TYPE ST_Software_Info :
STRUCT
	sTwinCATVersion		: STRING;
	iADSPort			: UINT;
	sProjectName		: STRING;
	sAppTimeStamp		: DATE_AND_TIME;
	rRealTimeUsage		: REAL;
	rRealTimeLatency	: REAL;
END_STRUCT
END_TYPE

(* stored: Version 1.1.0.1, ProductVersion 3.1.4022.18
   DUT ST_Software_Info: Id {e2f7158d-3a7b-4026-b26c-f43317a1f42e} *)
